(* LS Electric XG5000 project: hmi연동_실습 *)
(* PLC LSPLC *)

PROGRAM NewProgram (* task: 스캔 프로그램 *)
VAR
    INST4 : TP_UINT;
    R : BOOL;
END_VAR

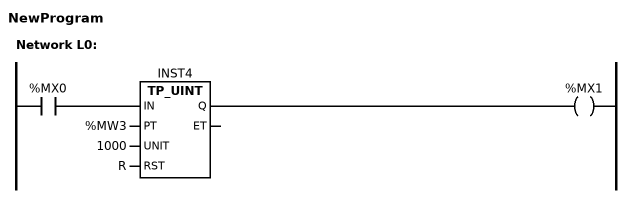
(* Rung L0 *)
INST4(IN := %MX0, PT := %MW3, UNIT := 1000, RST := R);
%MX1 := INST4.Q;
END_PROGRAM